Fanuc KAREL source: V_GET_PASSFL.kl

PROGRAM T
%NOLOCKGROUP
VAR
 v0 : STRING[40]
 v1 : INTEGER
 v2 : INTEGER
BEGIN
 V_GET_PASSFL(v0, v1, v2)
END T
